Fanuc KAREL source: kb00164.KL

-- PROVISIONAL review KL for V1013-1; original PC SHA256 02d273f96928f77f1d69f7878497fe29a76de8c46d30aee35e605397ff6e072b
-- Incomplete behavior may be omitted. Consult companion uncertainty JSON. Do not deploy.
PROGRAM KB00164
%NOLOCKGROUP
BEGIN
  -- UNRESOLVED_PC offsets 5-12; opcodes 9D,23
  -- UNRESOLVED_PC offsets 17-24; opcodes 9D,23
  -- UNRESOLVED_PC offsets 29-51; opcodes 27,22,22,22,31
  -- UNRESOLVED_PC offsets 56-60; opcodes 7F
END KB00164
